{attribute addProperty BoxType "EK1100-0000-0018"}
{attribute addProperty Id "Beckhoff_AMI8xxxEK1122Beckhoff_AMI8xxxEK1122_B38FD36B61276.5"}
{attribute addProperty CRC "1107672499"}
{attribute addProperty SizeInBites "612"}
{attribute addProperty SizeInBytes "76.5"}
TYPE EK1100_Beckhoff_AMI8xxx_4205BDB3 EXTENDS EK1100_179A0949 :
STRUCT
	{attribute addProperty Name "Beckhoff_AMI8xxxEK1122"}
	Beckhoff_AMI8xxxEK1122 : Beckhoff_AMI8xxxEK1122_B38FD36B;
END_STRUCT
END_TYPE

(* stored: Version 1.2.0.0, ProductVersion 3.1.4024.9
   DUT EK1100_Beckhoff_AMI8xxx_4205BDB3: Id {cfad1f6e-697f-42d2-96b0-663c8fc6a9d4} *)
